# EPICS StreamDevice protocol: EPICS/phoenixL300i.proto
OutTerminator = CR LF;
InTerminator = CR;
ReadTimeout = 100;
WriteTimeout = 100;
PollPeriod = 100;
ReplyTimeout = 1000;
LockTimeout = 5000;
ExtraInput = Ignore;

debug
{
	out "%s";
	in "%39c";
}

getStat
{
	out "*STAT?";
	in "%{INIT|ACCL|STBY|VENT|EVAC|MEAS|CAL|ERROR}";
}

readLeak
{
	out "*READ?";
	in "%e";
}

readLeakUnit
{
	out "*CONF:UNIT:LR?";
	in "%{mbar*l/s|Pa*m3/s|atm*cc/s|Torr*l/s}";
}

setLeakUnit
{
	out "*CONF:UNIT:LR %{MBAR*L/S|PA*M3/S|ATM*CC/S|TORR*L/S}";
	in "OK";
}

readPGPrs
{
	out "*MEAS:\$1?";
	in "%e";
}

setPGPrsUnit
{
	out "*CONF:UNIT:PRESSURE %{MBAR|ATM|PA|TORR}";
	in "OK";
}

readPGPrsUnit
{
	out "*CONF:UNIT:PRESSURE?";
	in "%{mbar|atm|Pa|Torr}";
}

setMode
{
	out "*%{Stop|Start|Vent|Purge|Cal|Zero}";
	in "OK";
}
